PROGRAM prgRWEffIO
VAR
	fbRW1		: FB_ReadWrite_V2;
	mFirst: BOOL;
END_VAR

fbRW1(bBusy=> , bError=> , udiErrorCodeOut=> , eErrorReadWrite_Out=> );


IF mFirst=FALSE THEN
	prgRWEffIO.fbRW1.eUploadType := 4;
	mFirst:=TRUE;	
END_IF

END_PROGRAM

(* stored: Version 1.1.0.1, ProductVersion 3.1.4024.11
   POU prgRWEffIO: Id {02288258-8b1d-4dbd-8ad3-1a1bf94c5849}, SpecialFunc None *)
